# EPICS autosave request: iocBoot/generic_motors_ioc/dbSave/GO_St_.req
%
% BURT Request File
%
% $(P)GO:St:  Goniometer support
%

file assy.req ASSY=$(P)GO:St
file mtr1.req MTR1=$(P)GO:msh
file mtr1.req MTR1=$(P)GO:msw
file mtr1.req MTR1=$(P)GO:msv
file drv1.req DRV1=$(P)GO:SH
file drv1.req DRV1=$(P)GO:SW
file drv1.req DRV1=$(P)GO:SV
